PROGRAM AutoMove3
VAR
END_VAR

END_PROGRAM

(* stored: Version 1.1.0.1, ProductVersion 3.1.4024.12
   POU AutoMove3: Id {d8ff9495-5edb-4363-8a3f-b0e10d5c02bf}, SpecialFunc None *)
